// TIA Portal V20 export
TYPE "AS-i esclavo"
   STRUCT
      Activo : Bool;
      Presente : Bool;
      Proyectado : Bool;
      Error : Bool;   // Esclavo con fallo de configuracion
      Reserved_1 : Bool;
      Reserved_2 : Bool;
      Reserved_3 : Bool;
      Reserved_4 : Bool;
      Reserved_5 : Bool;
      Reserved_6 : Bool;
      Reserved_7 : Bool;
      Reserved_8 : Bool;
      Reserved_9 : Bool;
      Reserved_10 : Bool;
      Reserved_11 : Bool;
      Reserved_12 : Bool;
   END_STRUCT;
END_TYPE
